TYPE UnitIndexerSlave EXTENDS UnitBase :
STRUCT
	guidMaster : DWORD;
END_STRUCT
END_TYPE

(* stored: Version 1.1.0.1, ProductVersion 3.1.4020.12
   DUT UnitIndexerSlave: Id {c804f68e-3486-40e4-8cee-cdf1b8928b7b} *)
